TYPE T_JsonDocumentString : STRING(Param_TcHaxx_Snappy.cMaxSizeJsonDocument); END_TYPE

(* stored: Version 1.1.0.1, ProductVersion 3.1.4024.12
   DUT T_JsonDocumentString: Id {4984266a-ac86-4849-b3c7-bf315bfd6dd3} *)
